(* IEC 61131-3 sources: volt/packages/volt-lsp-iec/test-corpus/pro2193/Device/Plc Logic/Application/09 Misc/Library Manager/CAA NetBaseSrv, 50 files *)

(* ---- CONNECTION_STATE.dut ---- *)
TYPE CONNECTION_STATE :
(
	CLOSED,
	ESTABLISHED,
	LISTEN,
	CLOSE_WAIT
);
END_TYPE

(* ---- E_ASYNC_OPERATION.dut ---- *)
TYPE E_ASYNC_OPERATION :
(
	NONE := 0,
	ABORT := 1,
	CYCLIC_ACT := 2
);
END_TYPE

(* ---- ERROR.dut ---- *)
TYPE ERROR :
(
	NO_ERROR := 0,
	FIRST_ERROR := 6000,
	TIME_OUT := 6001,
	INVALID_ADDR := 6002,
	INVALID_HANDLE := 6003,
	INVALID_DATAPOINTER := 6004,
	INVALID_DATASIZE := 6005,
	UDP_RECEIVE_ERROR := 6006,
	UDP_SEND_ERROR := 6007,
	UDP_SEND_NOT_COMPLETE := 6008,
	UDP_OPEN_ERROR := 6009,
	UDP_CLOSE_ERROR := 6010,
	TCP_SEND_ERROR := 6011,
	TCP_RECEIVE_ERROR := 6012,
	TCP_OPEN_ERROR := 6013,
	TCP_CONNECT_ERROR := 6014,
	TCP_CLOSE_ERROR := 6015,
	TCP_SERVER_ERROR := 6016,
	WRONG_PARAMETER := 6017,
	ERROR_UNKNOWN := 6018,
	TCP_NO_CONNECTION := 6019,
	IOCTL_ERROR := 6020,
	FIRST_MF := 6050,
	LAST_ERROR := 6099
);
END_TYPE

(* ---- IP_ADDR.dut ---- *)
TYPE IP_ADDR :
STRUCT
	SADDR : STRING(80);
END_STRUCT
END_TYPE

(* ---- NBS_TCP_CLIENT_OPEN_PARAMS.dut ---- *)
TYPE NBS_TCP_CLIENT_OPEN_PARAMS :
STRUCT
	UDITIMEOUT : UDINT;
	IPADDR : IP_ADDR;
	UIPORT : UINT;
	HCONNECTION : CAA.HANDLE;
	BYSTATE : BYTE;
END_STRUCT
END_TYPE

(* ---- NBS_TCP_CLOSE_PARAMS.dut ---- *)
TYPE NBS_TCP_CLOSE_PARAMS :
STRUCT
	HSOCKET : CAA.HANDLE;
END_STRUCT
END_TYPE

(* ---- NBS_TCP_CONNECTION_OPEN_PARAMS.dut ---- *)
TYPE NBS_TCP_CONNECTION_OPEN_PARAMS :
STRUCT
	HSERVER : CAA.HANDLE;
	HCONNECTION : CAA.HANDLE;
END_STRUCT
END_TYPE

(* ---- NBS_TCP_READ_PARAMS.dut ---- *)
TYPE NBS_TCP_READ_PARAMS :
STRUCT
	HCONNECTION : CAA.HANDLE;
	SZSIZE : CAA.SIZE;
	XREADY : BOOL;
	HBUFFER : CAA.HANDLE;
END_STRUCT
END_TYPE

(* ---- NBS_TCP_SERVER_OPEN_PARAMS.dut ---- *)
TYPE NBS_TCP_SERVER_OPEN_PARAMS :
STRUCT
	IPADDR : IP_ADDR;
	UIPORT : UINT;
	HSERVER : CAA.HANDLE;
END_STRUCT
END_TYPE

(* ---- NBS_TCP_WRITE_PARAMS.dut ---- *)
TYPE NBS_TCP_WRITE_PARAMS :
STRUCT
	HCONNECTION : CAA.HANDLE;
	HBUFFER : CAA.HANDLE;
END_STRUCT
END_TYPE

(* ---- NBS_UDP_PEER_CLOSE_PARAMS.dut ---- *)
TYPE NBS_UDP_PEER_CLOSE_PARAMS :
STRUCT
	HPEER : CAA.HANDLE;
END_STRUCT
END_TYPE

(* ---- NBS_UDP_PEER_OPEN_PARAMS.dut ---- *)
TYPE NBS_UDP_PEER_OPEN_PARAMS :
STRUCT
	IPADDR : IP_ADDR;
	UIPORT : UINT;
	IPMULTICAST : IP_ADDR;
	HPEER : CAA.HANDLE;
END_STRUCT
END_TYPE

(* ---- NBS_UDP_RECEIVE_PARAMS.dut ---- *)
TYPE NBS_UDP_RECEIVE_PARAMS :
STRUCT
	HPEER : CAA.HANDLE;
	SZSIZE : CAA.SIZE;
	XREADY : BOOL;
	IPFROM : IP_ADDR;
	UIPORTFROM : UINT;
	HBUFFER : CAA.HANDLE;
END_STRUCT
END_TYPE

(* ---- NBS_UDP_SEND_PARAMS.dut ---- *)
TYPE NBS_UDP_SEND_PARAMS :
STRUCT
	HPEER : CAA.HANDLE;
	IPADDR : IP_ADDR;
	UIPORT : UINT;
	HBUFFER : CAA.HANDLE;
END_STRUCT
END_TYPE

(* ---- SERVER_STATE.dut ---- *)
TYPE SERVER_STATE :
(
	SERVER_OPEN_INIT := 1,
	EXECUTE_SERVER_OPEN := 2,
	LISTENING := 3,
	EXECUTE_SERVER_CLOSE := 4,
	NOT_LISTENING := 5
);
END_TYPE

(* ---- ST_ASYNC.dut ---- *)
TYPE ST_ASYNC :
STRUCT
	HJOB : RTS_IEC_HANDLE := RTS_INVALID_HANDLE;
	UDISTATE : UDINT := ASYNCSTATE_READY;
	RESULT : RTS_IEC_RESULT;
	ASYNCJOBPARAM : ASYNCJOB_PARAM;
	CURRENTOP : E_ASYNC_OPERATION := E_ASYNC_OPERATION.NONE;
END_STRUCT
END_TYPE

(* ---- TCP_WRITE_STATE.dut ---- *)
TYPE TCP_WRITE_STATE :
(
	IDLE := 0,
	SENDING,
	DONE
);
END_TYPE

(* ---- ASYNCGLOB.gvl ---- *)
VAR_GLOBAL
	G_XGLOBALLIBINITDONE : BOOL := AsyncInitTask();
	GC_STASKRW : STRING := 'CAA_NetBaseServices_RW';
	GC_STASKOPENER : STRING := gc_sTaskRW;
END_VAR

(* ---- CAA_ASM_CONSTANTS.gvl ---- *)
VAR_GLOBAL
	UDP_PEER_OPEN_JOB_ID : UDINT := 16#50001;
	UDP_PEER_CLOSE_JOB_ID : UDINT := 16#50002;
	UDP_RECEIVE_JOB_ID : UDINT := 16#50003;
	UDP_SEND_JOB_ID : UDINT := 16#50004;
	TCP_SERVER_OPEN_JOB_ID : UDINT := 16#50005;
	TCP_CLIENT_OPEN_JOB_ID : UDINT := 16#50006;
	TCP_CONNECTION_OPEN_JOB_ID : UDINT := 16#50007;
	TCP_CLOSE_JOB_ID : UDINT := 16#50008;
	TCP_READ_JOB_ID : UDINT := 16#50009;
	TCP_WRITE_JOB_ID : UDINT := 16#5000A;
END_VAR

(* ---- CONSTANTS.gvl ---- *)
VAR_GLOBAL
	GC_FIRST_MULTICAST_IP : UDINT := 16#E0000000;
	GC_LAST_MULTICAST_IP : UDINT := 16#EFFFFFFF;
END_VAR

(* ---- FUNCTIONALITIES.gvl ---- *)
VAR_GLOBAL
	GC_XSUPPORTSTCPCLIENTSETADAPTER : BOOL;
END_VAR

(* ---- HOTO.gvl ---- *)
VAR_GLOBAL
	IDUMMY : INT;
END_VAR

(* ---- PARAM.gvl ---- *)
VAR_GLOBAL
	GC_UDITASKRWPRIORITY : UDINT := 240;
	GC_UDITASKOPENERPRIORITY : UDINT := gc_udiTaskRWPriority;
END_VAR

(* ---- VARIABLES.gvl ---- *)
VAR_GLOBAL
	G_HSOCKETCLASS : CAA.HANDLE;
END_VAR

(* ---- VERSIONCONSTANTS.gvl ---- *)
VAR_GLOBAL
	GC_BYVERSION : BYTE := 1;
	GC_BYVERSION_1 : BYTE := 0;
END_VAR

(* ---- ITCPCONNECTION.itf ---- *)
INTERFACE ITCPCONNECTION
END_INTERFACE

METHOD PRVCLOSE : ERROR
VAR_INPUT
	XDUMMY : BOOL;
END_VAR
END_METHOD

METHOD PRVESTABLISH : ERROR
END_METHOD

(* ---- ITCPSERVER.itf ---- *)
INTERFACE ITCPSERVER
END_INTERFACE

METHOD PRVADDCONNECTION : ERROR
VAR_INPUT
	CONNECTION : ITCPConnection;
END_VAR
END_METHOD

METHOD PRVREMOVECONNECTION : ERROR
VAR_INPUT
	CONNECTION : ITCPConnection;
END_VAR
END_METHOD

(* ---- ASYNCINITTASK.pou ---- *)
FUNCTION ASYNCINITTASK : BOOL
END_FUNCTION

(* ---- ASYNCINITTASK2INIT.pou ---- *)
FUNCTION ASYNCINITTASK2INIT : RTS_IEC_RESULT
VAR_INPUT
	PPARAM : __XWORD;
END_VAR
END_FUNCTION

(* ---- DUMMYJOB.pou ---- *)
FUNCTION DUMMYJOB : RTS_IEC_RESULT
VAR_INPUT
	PPARAM : __XWORD;
END_VAR
END_FUNCTION

(* ---- GETSUPPLIERVERSION.pou ---- *)
FUNCTION GETSUPPLIERVERSION : WORD
END_FUNCTION

(* ---- GETTCPSOCKETHANDLE.pou ---- *)
FUNCTION GETTCPSOCKETHANDLE : SysTypes.RTS_IEC_HANDLE
VAR_INPUT
	HCONNECTION : CAA.HANDLE;
END_VAR
END_FUNCTION

(* ---- GETUDPSOCKETHANDLE.pou ---- *)
FUNCTION GETUDPSOCKETHANDLE : SysTypes.RTS_IEC_HANDLE
VAR_INPUT
	HPEER : CAA.HANDLE;
END_VAR
END_FUNCTION

(* ---- IPSTRING_TO_UDINT.pou ---- *)
FUNCTION IPSTRING_TO_UDINT : UDINT
VAR_INPUT
	SIPADDRESS : STRING;
END_VAR
END_FUNCTION

(* ---- IS_MULTICAST_GROUP.pou ---- *)
FUNCTION IS_MULTICAST_GROUP : BOOL
VAR_INPUT
	UDIIPADDRESS : UDINT;
END_VAR
END_FUNCTION

(* ---- UDINT_TO_IPSTRING.pou ---- *)
FUNCTION UDINT_TO_IPSTRING : STRING
VAR_INPUT
	UDIIPADDRESS : UDINT;
END_VAR
END_FUNCTION

(* ---- UDP_GETDATASIZE.pou ---- *)
FUNCTION UDP_GETDATASIZE : CAA.SIZE
VAR_INPUT
	HPEER : CAA.HANDLE;
	PEERROR : POINTER TO ERROR;
END_VAR
END_FUNCTION

(* ---- TCP_CLIENT.pou ---- *)
FUNCTION_BLOCK TCP_CLIENT EXTENDS LTrig
VAR_INPUT
	UDITIMEOUT : UDINT := 0;
	IPADDR : IP_ADDR;
	UIPORT : UINT;
END_VAR
VAR_OUTPUT
	EERROR : ERROR;
	XACTIVE : BOOL;
	HCONNECTION : CAA.HANDLE;
END_VAR
VAR
	_UIPORT : UINT;
	_IPADDR : IP_ADDR;
	_ITFCONNECTION : TCPConnection;
	_TKSTART : CAA.TICK;
	_TCPCONNECTOR : TCP.Connector;
	_REBUILDDETECTRISINGEDGE : BOOL := FALSE;
	_ASYNC : ST_ASYNC;
	_ASYNCCLOSER : ST_ASYNC;
	_ASYNCRESETOUTPUTS : ST_ASYNC;
	_DBHOLDVALVS1TICK : BOOL;
	_DB_XDONE : BOOL;
	_DB_XBUSY : BOOL;
	_DB_XERROR : BOOL;
	_DB_IERROR : INT;
	_DB_EERROR : ERROR;
	_DB_XACTIVE : BOOL;
	_DB_HCONNECTION : CAA.HANDLE;
END_VAR
END_FUNCTION_BLOCK

METHOD FB_EXIT : BOOL
VAR_INPUT
	BINCOPYCODE : BOOL;
END_VAR
END_METHOD

METHOD FB_INIT : BOOL
VAR_INPUT
	BINITRETAINS : BOOL;
	BINCOPYCODE : BOOL;
END_VAR
END_METHOD

METHOD SETADAPTER : ERROR
VAR_INPUT
	IPADDR : IP_ADDR;
END_VAR
END_METHOD

METHOD PRVABORT : BOOL
END_METHOD

METHOD PRVASYNCABORT : RTS_IEC_RESULT
VAR_INPUT
	PPARAM : __XWORD;
END_VAR
END_METHOD

METHOD PRVASYNCCYCLICACTION : RTS_IEC_RESULT
VAR_INPUT
	PPARAM : __XWORD;
END_VAR
END_METHOD

METHOD PRVASYNCRESETOUTPUTS : RTS_IEC_RESULT
VAR_INPUT
	PPARAM : __XWORD;
END_VAR
END_METHOD

METHOD PRVCLOSE : BOOL
END_METHOD

METHOD PRVCYCLICACTION : BOOL
END_METHOD

METHOD PRVRESETOUTPUTS : BOOL
END_METHOD

METHOD PRVSTART : BOOL
END_METHOD

(* ---- TCP_CONNECTION.pou ---- *)
FUNCTION_BLOCK TCP_CONNECTION EXTENDS LTrig
VAR_INPUT
	HSERVER : CAA.HANDLE;
END_VAR
VAR_OUTPUT
	EERROR : ERROR;
	XACTIVE : BOOL;
	HCONNECTION : CAA.HANDLE;
END_VAR
VAR
	HCONNECTIONTMP : CAA.HANDLE;
	ITFSERVER : ITCPServer;
	PSERVER : POINTER TO TCP_Server;
	IINPUTERROR : ERROR;
	ITFCONNECTION : TCPConnection;
	_ASYNC : ST_ASYNC;
	_ASYNCCLOSER : ST_ASYNC;
	_ASYNCRESETOUTPUTS : ST_ASYNC;
	_REBUILDDETECTRISINGEDGE : BOOL := FALSE;
	_DBHOLDVALVS1TICK : BOOL;
	_DB_XDONE : BOOL;
	_DB_XBUSY : BOOL;
	_DB_XERROR : BOOL;
	_DB_IERROR : INT;
	_DB_EERROR : ERROR;
	_DB_XACTIVE : BOOL;
	_DB_HCONNECTION : CAA.HANDLE;
	IPADDRESS : SysSocket.INADDR;
END_VAR
END_FUNCTION_BLOCK

METHOD FB_EXIT : BOOL
VAR_INPUT
	BINCOPYCODE : BOOL;
END_VAR
END_METHOD

METHOD FB_INIT : BOOL
VAR_INPUT
	BINITRETAINS : BOOL;
	BINCOPYCODE : BOOL;
END_VAR
END_METHOD

METHOD PRVABORT : BOOL
END_METHOD

METHOD PRVASYNCABORT : RTS_IEC_RESULT
VAR_INPUT
	PPARAM : __XWORD;
END_VAR
END_METHOD

METHOD PRVASYNCCYCLICACTION : RTS_IEC_RESULT
VAR_INPUT
	PPARAM : __XWORD;
END_VAR
END_METHOD

METHOD PRVASYNCRESETOUTPUTS : RTS_IEC_RESULT
VAR_INPUT
	PPARAM : __XWORD;
END_VAR
END_METHOD

METHOD PRVCLOSE : BOOL
END_METHOD

METHOD PRVCYCLICACTION : BOOL
END_METHOD

METHOD PRVRESETOUTPUTS : BOOL
END_METHOD

METHOD PRVSTART : BOOL
END_METHOD

(* ---- TCP_READ.pou ---- *)
FUNCTION_BLOCK TCP_READ EXTENDS LTrig
VAR_INPUT
	HCONNECTION : CAA.HANDLE;
	SZSIZE : CAA.SIZE;
	PDATA : CAA.PVOID;
END_VAR
VAR_OUTPUT
	EERROR : ERROR;
	XREADY : BOOL;
	SZCOUNT : CAA.SIZE;
END_VAR
VAR
	IINPUTERROR : ERROR;
	ITFCONNECTION : ITCPConnection;
	_ASYNC : ST_ASYNC;
	_DBHOLDVALVS1TICK : BOOL;
	_DB_XDONE : BOOL;
	_DB_XBUSY : BOOL;
	_DB_XERROR : BOOL;
	_DB_IERROR : INT;
	_DB_EERROR : ERROR;
	_DB_XREADY : BOOL;
	_DB_SZCOUNT : CAA.SIZE;
END_VAR
END_FUNCTION_BLOCK

METHOD FB_EXIT : BOOL
VAR_INPUT
	BINCOPYCODE : BOOL;
END_VAR
END_METHOD

METHOD FB_INIT : BOOL
VAR_INPUT
	BINITRETAINS : BOOL;
	BINCOPYCODE : BOOL;
END_VAR
END_METHOD

METHOD PRVABORT : BOOL
END_METHOD

METHOD PRVASYNCCYCLICACTION : RTS_IEC_RESULT
VAR_INPUT
	PPARAM : __XWORD;
END_VAR
END_METHOD

METHOD PRVCYCLICACTION : BOOL
END_METHOD

METHOD PRVRESETOUTPUTS : BOOL
END_METHOD

METHOD PRVSTART : BOOL
END_METHOD

(* ---- TCP_READBUFFER.pou ---- *)
FUNCTION_BLOCK TCP_READBUFFER EXTENDS LTrig
VAR_INPUT
	HCONNECTION : CAA.HANDLE;
END_VAR
VAR_OUTPUT
	EERROR : ERROR;
	XREADY : BOOL;
	HBUFFER : CAA.HANDLE;
END_VAR
VAR
	IINPUTERROR : ERROR;
	ITFCONNECTION : ITCPConnection;
	_ASYNC : ST_ASYNC;
	_DBHOLDVALVS1TICK : BOOL;
	_DB_XDONE : BOOL;
	_DB_XBUSY : BOOL;
	_DB_XERROR : BOOL;
	_DB_IERROR : INT;
	_DB_EERROR : ERROR;
	_DB_XREADY : BOOL;
	_DB_HBUFFER : CAA.HANDLE;
END_VAR
END_FUNCTION_BLOCK

METHOD FB_EXIT : BOOL
VAR_INPUT
	BINCOPYCODE : BOOL;
END_VAR
END_METHOD

METHOD FB_INIT : BOOL
VAR_INPUT
	BINITRETAINS : BOOL;
	BINCOPYCODE : BOOL;
END_VAR
END_METHOD

METHOD PRVABORT : BOOL
END_METHOD

METHOD PRVASYNCCYCLICACTION : RTS_IEC_RESULT
VAR_INPUT
	PPARAM : __XWORD;
END_VAR
END_METHOD

METHOD PRVCYCLICACTION : BOOL
END_METHOD

METHOD PRVRESETOUTPUTS : BOOL
END_METHOD

METHOD PRVSTART : BOOL
END_METHOD

(* ---- TCP_SERVER.pou ---- *)
FUNCTION_BLOCK TCP_SERVER EXTENDS LTrig
VAR_INPUT
	IPADDR : IP_ADDR := STRUCT(sAddr := '0.0.0.0');
	UIPORT : UINT;
END_VAR
VAR_OUTPUT
	EERROR : ERROR;
	HSERVER : CAA.HANDLE;
END_VAR
VAR
	_UIPORT : UINT;
	_IPADDR : IP_ADDR;
	_LSTCONNECTIONS : LAT.List;
	_ITFSERVER : ITCPServer;
	_PSERVER : POINTER TO TCP_Server;
	_TCPLISTENER : TCP.Listener;
	_ESTATE : SERVER_STATE := SERVER_STATE.NOT_LISTENING;
	_REBUILDDETECTRISINGEDGE : BOOL := FALSE;
	_ASYNC : ST_ASYNC;
	_ASYNCCLOSER : ST_ASYNC;
	_ASYNCRESETOUTPUTS : ST_ASYNC;
	_DBHOLDVALVS1TICK : BOOL;
	_DB_XDONE : BOOL;
	_DB_XBUSY : BOOL;
	_DB_XERROR : BOOL;
	_DB_IERROR : INT;
	_DB_EERROR : ERROR;
	_DB_HSERVER : CAA.HANDLE;
END_VAR
END_FUNCTION_BLOCK

METHOD FB_EXIT : BOOL
VAR_INPUT
	BINCOPYCODE : BOOL;
END_VAR
END_METHOD

METHOD FB_INIT : BOOL
VAR_INPUT
	BINITRETAINS : BOOL;
	BINCOPYCODE : BOOL;
END_VAR
END_METHOD

METHOD PRVABORT : BOOL
END_METHOD

METHOD PRVADDCONNECTION : ERROR
VAR_INPUT
	CONNECTION : ITCPConnection;
END_VAR
END_METHOD

METHOD PRVASYNCABORT : RTS_IEC_RESULT
VAR_INPUT
	PPARAM : __XWORD;
END_VAR
END_METHOD

METHOD PRVASYNCCYCLICACTION : RTS_IEC_RESULT
VAR_INPUT
	PPARAM : __XWORD;
END_VAR
END_METHOD

METHOD PRVASYNCRESETOUTPUTS : RTS_IEC_RESULT
VAR_INPUT
	PPARAM : __XWORD;
END_VAR
END_METHOD

METHOD PRVCLOSE
END_METHOD

METHOD PRVCYCLICACTION : BOOL
END_METHOD

METHOD PRVREMOVECONNECTION : ERROR
VAR_INPUT
	CONNECTION : ITCPConnection;
END_VAR
END_METHOD

METHOD PRVRESETOUTPUTS : BOOL
END_METHOD

METHOD PRVSTART : BOOL
END_METHOD

(* ---- TCP_WRITE.pou ---- *)
FUNCTION_BLOCK TCP_WRITE EXTENDS ETrigTo
VAR_INPUT
	HCONNECTION : CAA.HANDLE;
	SZSIZE : CAA.SIZE;
	PDATA : CAA.PVOID;
END_VAR
VAR_OUTPUT
	EERROR : ERROR;
END_VAR
VAR
	ESEGBUFMANERROR : SBM.ERROR;
	IINPUTERROR : ERROR;
	ITFCONNECTION : ITCPConnection;
	_SZSENTBYTES : CAA.SIZE;
	_EWRITESTATE : TCP_WRITE_STATE;
	_ASYNC : ST_ASYNC;
	_ASYNCCLOSER : ST_ASYNC;
	_ASYNCRESETOUTPUTS : ST_ASYNC;
	_DBHOLDVALVS1TICK : BOOL;
	_DB_XDONE : BOOL;
	_DB_XBUSY : BOOL;
	_DB_XERROR : BOOL;
	_DB_IERROR : INT;
	_DB_EERROR : ERROR;
END_VAR
END_FUNCTION_BLOCK

METHOD FB_EXIT : BOOL
VAR_INPUT
	BINCOPYCODE : BOOL;
END_VAR
END_METHOD

METHOD FB_INIT : BOOL
VAR_INPUT
	BINITRETAINS : BOOL;
	BINCOPYCODE : BOOL;
END_VAR
END_METHOD

METHOD PRVABORT : BOOL
END_METHOD

METHOD PRVASYNCABORT : RTS_IEC_RESULT
VAR_INPUT
	PPARAM : __XWORD;
END_VAR
END_METHOD

METHOD PRVASYNCCYCLICACTION : RTS_IEC_RESULT
VAR_INPUT
	PPARAM : __XWORD;
END_VAR
END_METHOD

METHOD PRVCYCLICACTION : BOOL
END_METHOD

METHOD PRVRESETOUTPUTS : BOOL
END_METHOD

METHOD PRVSTART : BOOL
END_METHOD

(* ---- TCP_WRITEBUFFER.pou ---- *)
FUNCTION_BLOCK TCP_WRITEBUFFER EXTENDS ETrigTo
VAR_INPUT
	HCONNECTION : CAA.HANDLE;
	HBUFFER : CAA.HANDLE;
END_VAR
VAR_OUTPUT
	EERROR : ERROR;
END_VAR
VAR
	_HBUFFER : CAA.HANDLE;
	IINPUTERROR : ERROR;
	ITFCONNECTION : ITCPConnection;
	_SZSENTBYTES : CAA.SIZE;
	_EWRITESTATE : TCP_WRITE_STATE;
	_ASYNC : ST_ASYNC;
	_ASYNCCLOSER : ST_ASYNC;
	_ASYNCRESETOUTPUTS : ST_ASYNC;
	_DBHOLDVALVS1TICK : BOOL;
	_DB_XDONE : BOOL;
	_DB_XBUSY : BOOL;
	_DB_XERROR : BOOL;
	_DB_IERROR : INT;
	_DB_EERROR : ERROR;
END_VAR
END_FUNCTION_BLOCK

METHOD FB_EXIT : BOOL
VAR_INPUT
	BINCOPYCODE : BOOL;
END_VAR
END_METHOD

METHOD FB_INIT : BOOL
VAR_INPUT
	BINITRETAINS : BOOL;
	BINCOPYCODE : BOOL;
END_VAR
END_METHOD

METHOD PRVABORT : BOOL
END_METHOD

METHOD PRVASYNCABORT : RTS_IEC_RESULT
VAR_INPUT
	PPARAM : __XWORD;
END_VAR
END_METHOD

METHOD PRVASYNCCYCLICACTION : RTS_IEC_RESULT
VAR_INPUT
	PPARAM : __XWORD;
END_VAR
END_METHOD

METHOD PRVASYNCRESETOUTPUTS : RTS_IEC_RESULT
VAR_INPUT
	PPARAM : __XWORD;
END_VAR
END_METHOD

METHOD PRVCYCLICACTION : BOOL
END_METHOD

METHOD PRVRESETOUTPUTS : BOOL
END_METHOD

METHOD PRVSTART : BOOL
END_METHOD

(* ---- TCPCONNECTION.pou ---- *)
FUNCTION_BLOCK TCPCONNECTION EXTENDS Element
VAR
	TCPSTREAM : TCP.Stream;
	HSOCKET : SysTypes.RTS_IEC_HANDLE := SysTypes.RTS_INVALID_HANDLE;
	ESTATE : CONNECTION_STATE := CONNECTION_STATE.LISTEN;
	_PUSHBACK1READBYTE_DATA : BYTE;
	_PUSHBACK1READBYTE_CALLED : BOOL;
	PRVSOCKETHANDLE : RTS_IEC_HANDLE;
	PRVSTATE : CONNECTION_STATE;
	PRVSTREAM : POINTER TO TCP.Stream;
END_VAR
END_FUNCTION_BLOCK

METHOD FB_EXIT : BOOL
VAR_INPUT
	BINCOPYCODE : BOOL;
END_VAR
END_METHOD

METHOD SETPUSHBACK1READBYTE
VAR_INPUT
	DATA : BYTE;
	CALLED : BOOL;
END_VAR
END_METHOD

METHOD PRVCLOSE : ERROR
VAR_INPUT
	XDUMMY : BOOL;
END_VAR
END_METHOD

METHOD PRVESTABLISH : ERROR
END_METHOD

(* ---- UDP_PEER.pou ---- *)
FUNCTION_BLOCK UDP_PEER EXTENDS LTrig
VAR_INPUT
	IPADDR : IP_ADDR := STRUCT(sAddr := '0.0.0.0');
	UIPORT : UINT;
	IPMULTICAST : IP_ADDR := STRUCT(sAddr := '255.255.255.255');
END_VAR
VAR_OUTPUT
	EERROR : ERROR;
	XACTIVE : BOOL;
	HPEER : CAA.HANDLE;
END_VAR
VAR
	_UDIIPADDRESS : UDINT;
	_UDIMCIPADDRESS : UDINT;
	_UDPDRIVER : UDP.UDPDriver;
	_UDPPORT : UDP.Port;
END_VAR
END_FUNCTION_BLOCK

METHOD FB_EXIT : BOOL
VAR_INPUT
	BINCOPYCODE : BOOL;
END_VAR
END_METHOD

METHOD PRVABORT : BOOL
END_METHOD

METHOD PRVCLOSE
END_METHOD

METHOD PRVCYCLICACTION : BOOL
END_METHOD

METHOD PRVRESETOUTPUTS : BOOL
END_METHOD

METHOD PRVSTART : BOOL
END_METHOD

(* ---- UDP_RECEIVE.pou ---- *)
FUNCTION_BLOCK UDP_RECEIVE EXTENDS LTrig
VAR_INPUT
	HPEER : CAA.HANDLE;
	SZSIZE : CAA.SIZE;
	PDATA : CAA.PVOID;
END_VAR
VAR_OUTPUT
	EERROR : ERROR;
	XREADY : BOOL;
	IPFROM : IP_ADDR;
	UIPORTFROM : UINT;
	SZCOUNT : CAA.SIZE;
END_VAR
VAR
	_PUDPPORT : POINTER TO UDP.Port;
	IINPUTERROR : ERROR;
END_VAR
END_FUNCTION_BLOCK

METHOD PRVABORT : BOOL
END_METHOD

METHOD PRVCYCLICACTION : BOOL
END_METHOD

METHOD PRVRESETOUTPUTS : BOOL
END_METHOD

METHOD PRVSTART : BOOL
END_METHOD

(* ---- UDP_RECEIVEBUFFER.pou ---- *)
FUNCTION_BLOCK UDP_RECEIVEBUFFER EXTENDS LTrig
VAR_INPUT
	HPEER : CAA.HANDLE;
END_VAR
VAR_OUTPUT
	EERROR : ERROR;
	XREADY : BOOL;
	IPFROM : IP_ADDR;
	UIPORTFROM : UINT;
	HBUFFER : CAA.HANDLE;
END_VAR
VAR
	_PUDPPORT : POINTER TO UDP.Port;
	IINPUTERROR : ERROR;
END_VAR
END_FUNCTION_BLOCK

METHOD PRVABORT : BOOL
END_METHOD

METHOD PRVCYCLICACTION : BOOL
END_METHOD

METHOD PRVRESETOUTPUTS : BOOL
END_METHOD

METHOD PRVSTART : BOOL
END_METHOD

(* ---- UDP_SEND.pou ---- *)
FUNCTION_BLOCK UDP_SEND EXTENDS ETrigTo
VAR_INPUT
	HPEER : CAA.HANDLE;
	IPADDR : IP_ADDR;
	UIPORT : UINT;
	SZSIZE : CAA.SIZE;
	PDATA : CAA.PVOID;
END_VAR
VAR_OUTPUT
	EERROR : ERROR;
END_VAR
VAR
	IINPUTERROR : ERROR;
	_PUDPPORT : POINTER TO UDP.Port;
END_VAR
END_FUNCTION_BLOCK

METHOD PRVABORT : BOOL
END_METHOD

METHOD PRVCYCLICACTION : BOOL
END_METHOD

METHOD PRVRESETOUTPUTS : BOOL
END_METHOD

METHOD PRVSTART : BOOL
END_METHOD

(* ---- UDP_SENDBUFFER.pou ---- *)
FUNCTION_BLOCK UDP_SENDBUFFER EXTENDS ETrigTo
VAR_INPUT
	HPEER : CAA.HANDLE;
	IPADDR : IP_ADDR;
	UIPORT : UINT;
	HBUFFER : CAA.HANDLE;
END_VAR
VAR_OUTPUT
	EERROR : ERROR;
END_VAR
VAR
	_HBUFFER : CAA.HANDLE;
	IINPUTERROR : ERROR;
	_PUDPPORT : POINTER TO UDP.Port;
END_VAR
END_FUNCTION_BLOCK

METHOD FB_EXIT : BOOL
VAR_INPUT
	BINCOPYCODE : BOOL;
END_VAR
END_METHOD

METHOD PRVABORT : BOOL
END_METHOD

METHOD PRVCYCLICACTION : BOOL
END_METHOD

METHOD PRVRESETOUTPUTS : BOOL
END_METHOD

METHOD PRVSTART : BOOL
END_METHOD
